(* IEC 61131-3 sources: etrolProject/分输站, 3 files *)

(* ---- com1tx.ST ---- *)
PROGRAM com1tx
VAR_EXTERNAL

END_VAR

VAR_GLOBAL

END_VAR

VAR
i		   :  UINT;
ai0_val    :  REAL :=0.0;
ai1_val    :  REAL :=0.0;
ai2_val    :  REAL :=0.0;
ai3_val    :  REAL :=0.0;
ai4_val    :  REAL :=0.0;
ai5_val    :  REAL :=0.0;
ai6_val    :  REAL :=0.0;
ai7_val    :  REAL :=0.0;
ai8_val    :  REAL :=0.0;
ai9_val    :  REAL :=0.0;
ai10_val    :  REAL :=0.0;
ai11_val    :  REAL :=0.0;
addr_val	:  UINT;
button AT %I0.0		:	BOOL;
blinker AT %Q0.6 	:	BOOL;
adr_var : UINT;
val_var : UINT;
lock_var : UINT := 0;
duishe_var : UINT := 0;
jinkoup_var : REAL;
chukoup_var : REAL;
huanrewd_var : REAL;

REG_W_UINT_VAR : REG_W_UINT;
REG_R_UINT_VAR : REG_R_UINT;
REG_MOVE_VAR   : REG_MOVE;
REG_R_REAL_VAL : REG_R_REAL;
REG_W_REAL_VAL : REG_W_REAL;
END_VAR
(*压变，温变采集*)

addr_val := 30017;
REG_R_REAL_VAL(ADDR := addr_val, SWAP := 0);
ai0_val := (REG_R_REAL_VAL.DATA - 4.0)/16.0 * 10000.0;
addr_val := 40001;
REG_W_REAL_VAL(ADDR := addr_val, SWAP := 0, DATA := ai0_val);

addr_val := 30019;
REG_R_REAL_VAL(ADDR := addr_val, SWAP := 0);
ai0_val := (REG_R_REAL_VAL.DATA - 4.0)/16.0 * 120.0 - 40.0;
addr_val := 40003;
REG_W_REAL_VAL(ADDR := addr_val, SWAP := 0, DATA := ai0_val);

addr_val := 30021;
REG_R_REAL_VAL(ADDR := addr_val, SWAP := 0);
ai0_val := (REG_R_REAL_VAL.DATA - 4.0)/16.0 * 6000.0;
addr_val := 40005;
REG_W_REAL_VAL(ADDR := addr_val, SWAP := 0, DATA := ai0_val);

addr_val := 30023;
REG_R_REAL_VAL(ADDR := addr_val, SWAP := 0);
ai0_val := (REG_R_REAL_VAL.DATA - 4.0)/16.0 * 6000.0;
addr_val := 40007;
REG_W_REAL_VAL(ADDR := addr_val, SWAP := 0, DATA := ai0_val);

addr_val := 30025;
REG_R_REAL_VAL(ADDR := addr_val, SWAP := 0);
ai0_val := (REG_R_REAL_VAL.DATA - 4.0)/16.0 * 6000.0;
addr_val := 40009;
REG_W_REAL_VAL(ADDR := addr_val, SWAP := 0, DATA := ai0_val);

addr_val := 30027;
REG_R_REAL_VAL(ADDR := addr_val, SWAP := 0);
ai0_val := (REG_R_REAL_VAL.DATA - 4.0)/16.0 * 6000.0;
addr_val := 40011;
REG_W_REAL_VAL(ADDR := addr_val, SWAP := 0, DATA := ai0_val);

addr_val := 30029;
REG_R_REAL_VAL(ADDR := addr_val, SWAP := 0);
ai0_val := (REG_R_REAL_VAL.DATA - 4.0)/16.0 * 6000.0;
addr_val := 40013;
REG_W_REAL_VAL(ADDR := addr_val, SWAP := 0, DATA := ai0_val);

addr_val := 30031;
REG_R_REAL_VAL(ADDR := addr_val, SWAP := 0);
ai0_val := (REG_R_REAL_VAL.DATA - 4.0)/16.0 * 120.0 - 40.0;
addr_val := 40015;
REG_W_REAL_VAL(ADDR := addr_val, SWAP := 0, DATA := ai0_val);

addr_val := 30033;
REG_R_REAL_VAL(ADDR := addr_val, SWAP := 0);
ai0_val := (REG_R_REAL_VAL.DATA - 4.0)/16.0 * 100.0;
addr_val := 40089;
REG_W_REAL_VAL(ADDR := addr_val, SWAP := 0, DATA := ai0_val);

addr_val := 30035;
REG_R_REAL_VAL(ADDR := addr_val, SWAP := 0);
ai0_val := (REG_R_REAL_VAL.DATA - 4.0)/16.0 * 100.0;
addr_val := 40101;
REG_W_REAL_VAL(ADDR := addr_val, SWAP := 0, DATA := ai0_val);

addr_val := 30037;
REG_R_REAL_VAL(ADDR := addr_val, SWAP := 0);
ai0_val := (REG_R_REAL_VAL.DATA - 4.0)/16.0 * 100.0;
addr_val := 40017;
REG_W_REAL_VAL(ADDR := addr_val, SWAP := 0, DATA := ai0_val);

addr_val := 30039;
REG_R_REAL_VAL(ADDR := addr_val, SWAP := 0);
ai0_val := (REG_R_REAL_VAL.DATA - 4.0)/16.0 * 100.0;
addr_val := 40019;
REG_W_REAL_VAL(ADDR := addr_val, SWAP := 0, DATA := ai0_val);

addr_val := 30041;
REG_R_REAL_VAL(ADDR := addr_val, SWAP := 0);
ai0_val := (REG_R_REAL_VAL.DATA - 4.0)/16.0 * 500.0;
addr_val := 40115;
REG_W_REAL_VAL(ADDR := addr_val, SWAP := 0, DATA := ai0_val);

END_PROGRAM

(* ---- DIANJIARE.ST ---- *)
PROGRAM DIANJIARE
VAR_EXTERNAL

END_VAR

VAR_GLOBAL

END_VAR

VAR
blinker AT %Q0.0 	:	BOOL;
blinker2 AT %Q0.1 	:	BOOL;
blinker3 AT %Q0.2   :   BOOL;
blinker4 AT %Q0.3   :   BOOL;
blinker5 AT %Q0.4   :   BOOL;
blinker6 AT %Q0.5   :   BOOL;
blinker7 AT %Q0.6   :   BOOL;
blinker8 AT %Q0.7   :   BOOL;
blinker9 AT %Q1.0   :   BOOL;
blinker10 AT %Q1.1   :   BOOL;
blinker11 AT %Q1.2   :   BOOL;
blinker12 AT %Q1.3   :   BOOL;
blinker13 AT %Q1.4   :   BOOL;
jtbutton : uint;
sgbj : uint;
i : uint;
j : uint;
kdw : uint;
gdw :uint;
kdw2 : uint;
gdw2 :uint;
kdw3 : uint;
gdw3 :uint;
kdw4 : uint;
gdw4 :uint;
jt_gdw1 : uint;
jt_gdw2 : uint;
jt_kdw1 : uint;
jt_kdw2 : uint;
addr_val : uint;
wds_val : REAL;
wdx_val : REAL;
wd_val : REAL;
par_var : uint;
lock_var : uint;
jf_open : uint;
jf_close : uint;
jf2_open : uint;
jf2_close : uint;
jf3_open : uint;
jf3_close : uint;
jf4_open : uint;
jf4_close : uint;
szd_var : uint;
REG_W_UINT_VAR : REG_W_UINT;
REG_R_UINT_VAR : REG_R_UINT;
REG_MOVE_VAR   : REG_MOVE;
REG_R_REAL_VAL : REG_R_REAL;
REG_W_REAL_VAL : REG_W_REAL;
END_VAR

REG_R_UINT_VAR(ADDR := 10018);
jtbutton := REG_R_UINT_VAR.DATA;
(*急停未按下，阀门操作*)
IF jtbutton=0 THEN
	blinker3 := TRUE;
	blinker9 := FALSE;
	blinker12 := FALSE;
	(*判断进站气液联动阀是否已修改*)
	REG_R_UINT_VAR(ADDR := 40074);
	par_var := REG_R_UINT_VAR.DATA;
	IF par_var=1 THEN
	(*参数修改*)
		REG_W_UINT_VAR(ADDR := 40074, DATA := 0);
		REG_R_UINT_VAR(ADDR := 40071);
		jf_open := REG_R_UINT_VAR.DATA;
		IF jf_open=1 THEN
			blinker := TRUE;
		ELSE
			blinker := FALSE;

		END_IF;

		REG_R_UINT_VAR(ADDR := 40072);
		jf_close := REG_R_UINT_VAR.DATA;
		IF jf_close=1 THEN
			blinker2 := TRUE;
		ELSE
			blinker2 := FALSE;
		END_IF;
	ELSE
	(*参数未修改*)
		;
	END_IF;

	REG_R_UINT_VAR(ADDR := 10003);
	kdw := REG_R_UINT_VAR.DATA;
	IF kdw=1 THEN
		blinker := FALSE;
	ELSE
		;
	END_IF;

	REG_R_UINT_VAR(ADDR := 10004);
	gdw := REG_R_UINT_VAR.DATA;
	IF gdw=1 THEN
		blinker2 := FALSE;
	ELSE
		;
	END_IF;
	(*出站电动阀*)
	REG_R_UINT_VAR(ADDR := 40078);
	par_var := REG_R_UINT_VAR.DATA;
	IF par_var=1 THEN
	(*参数修改*)
		REG_W_UINT_VAR(ADDR := 40078, DATA := 0);
		REG_R_UINT_VAR(ADDR := 40075);
		jf2_open := REG_R_UINT_VAR.DATA;
		IF jf2_open=1 THEN
			blinker4 := TRUE;
		ELSE
			blinker4 := FALSE;

		END_IF;

		REG_R_UINT_VAR(ADDR := 40076);
		jf2_close := REG_R_UINT_VAR.DATA;
		IF jf2_close=1 THEN
			blinker5 := TRUE;
		ELSE
			blinker5 := FALSE;
		END_IF;
	ELSE
	(*参数未修改*)
		;
	END_IF;

	REG_R_UINT_VAR(ADDR := 10006);
	kdw2 := REG_R_UINT_VAR.DATA;
	IF kdw2=1 THEN
		blinker4 := FALSE;
	ELSE
		;
	END_IF;

	REG_R_UINT_VAR(ADDR := 10007);
	gdw2 := REG_R_UINT_VAR.DATA;
	IF gdw2=1 THEN
		blinker5 := FALSE;
	ELSE
		;
	END_IF;

	(*进站放空阀*)
	REG_R_UINT_VAR(ADDR := 40082);
	par_var := REG_R_UINT_VAR.DATA;
	IF par_var=1 THEN
	(*参数修改*)
		REG_W_UINT_VAR(ADDR := 40082, DATA := 0);
		REG_R_UINT_VAR(ADDR := 40079);
		jf3_open := REG_R_UINT_VAR.DATA;
		IF jf3_open=1 THEN
			blinker7 := TRUE;
		ELSE
			blinker7 := FALSE;

		END_IF;

		REG_R_UINT_VAR(ADDR := 40080);
		jf3_close := REG_R_UINT_VAR.DATA;
		IF jf3_close=1 THEN
			blinker8 := TRUE;
		ELSE
			blinker8 := FALSE;
		END_IF;
	ELSE
	(*参数未修改*)
		;
	END_IF;

	REG_R_UINT_VAR(ADDR := 10010);
	kdw3 := REG_R_UINT_VAR.DATA;
	IF kdw3=1 THEN
		blinker7 := FALSE;
	ELSE
		;
	END_IF;

	REG_R_UINT_VAR(ADDR := 10011);
	gdw3 := REG_R_UINT_VAR.DATA;
	IF gdw3=1 THEN
		blinker8 := FALSE;
	ELSE
		;
	END_IF;

	(*出站放空阀*)
	REG_R_UINT_VAR(ADDR := 40086);
	par_var := REG_R_UINT_VAR.DATA;
	IF par_var=1 THEN
	(*参数修改*)
		REG_W_UINT_VAR(ADDR := 40086, DATA := 0);
		REG_R_UINT_VAR(ADDR := 40083);
		jf4_open := REG_R_UINT_VAR.DATA;
		IF jf4_open=1 THEN
			blinker10 := TRUE;
		ELSE
			blinker10 := FALSE;

		END_IF;

		REG_R_UINT_VAR(ADDR := 40084);
		jf4_close := REG_R_UINT_VAR.DATA;
		IF jf4_close=1 THEN
			blinker11 := TRUE;
		ELSE
			blinker11 := FALSE;
		END_IF;
	ELSE
	(*参数未修改*)
		;
	END_IF;

	REG_R_UINT_VAR(ADDR := 10014);
	kdw4 := REG_R_UINT_VAR.DATA;
	IF kdw4=1 THEN
		blinker10 := FALSE;
	ELSE
		;
	END_IF;

	REG_R_UINT_VAR(ADDR := 10015);
	gdw4 := REG_R_UINT_VAR.DATA;
	IF gdw4=1 THEN
		blinker11 := FALSE;
	ELSE
		;
	END_IF;
ELSE
	(*急停关阀操作*)
	(*先关进站气液，出站电动，再开进出放空*)
	blinker3 := FALSE;
	blinker9 := TRUE;
	blinker12 := TRUE;
	REG_R_UINT_VAR(ADDR := 10004);
	jt_gdw1 := REG_R_UINT_VAR.DATA;
(*	IF jt_gdw1=1 THEN
		blinker2 := FALSE;
	ELSE
		blinker2 := TRUE;
	END_IF;
	*)
	REG_R_UINT_VAR(ADDR := 10007);
	jt_gdw2 := REG_R_UINT_VAR.DATA;
	IF jt_gdw2=1 THEN
		blinker5 := FALSE;
	ELSE
		blinker5 := TRUE;
	END_IF;

	IF jt_gdw1=1 AND jt_gdw2=1 THEN
		(*REG_R_UINT_VAR(ADDR := 10010);
		jt_kdw1 := REG_R_UINT_VAR.DATA;
		IF jt_kdw1=1 THEN
			blinker7 := FALSE;
		ELSE
			blinker7 := TRUE;
		END_IF;

		REG_R_UINT_VAR(ADDR := 10014);
		jt_kdw2 := REG_R_UINT_VAR.DATA;
		IF jt_kdw2=1 THEN
			blinker10 := FALSE;
		ELSE
			blinker10 := TRUE;
		END_IF;*)
		;
	ELSE
		;
	END_IF;
END_IF;

REG_R_UINT_VAR(ADDR := 40112);
par_var := REG_R_UINT_VAR.DATA;
IF par_var=1 THEN
	REG_W_UINT_VAR(ADDR := 40112, DATA := 0);
	REG_R_UINT_VAR(ADDR := 40111);
	sgbj := REG_R_UINT_VAR.DATA;
	IF sgbj=1 THEN
		blinker13 := TRUE;
	ELSE
		blinker13 := FALSE;
	END_IF;
ELSE
	;
END_IF;
END_PROGRAM

(* ---- RX1.ST ---- *)
PROGRAM RX1
VAR_EXTERNAL
jiachou : udint;
flow_val : REAL;
start_val : uint;

END_VAR

VAR_GLOBAL
jiachou1 : udint:=0;
END_VAR

VAR
tjf_ya1_val : uint;
tjf2_ya1_val : uint;
tjf_kd1_val : uint;
tjf_ya2_val : uint;
tjf_kd2_val : uint;
i : uint;
j : uint;
blinker AT %Q0.4 	:	BOOL;
djr_start AT %Q1.5  :   BOOL;
djr_stop  AT %Q1.6  :   BOOL;
djr_par : uint;
dir_mode : uint;
dir_temp : uint;
djr_qd   : uint;
djr_tz   : uint;
djr_settemp : REAL;
dir_settemp_val : uint;
dir_fktemp : uint;
jiachounew : udint;
par_var :uint;
lock_var : uint;
szd_var	:uint;
addr_val : uint;
shunshi_val : REAL;
tongji_val : REAL;
sdyl : REAL;
sdyl_val :uint;
sdyl1 : REAL;
sdyl1_val :uint;
tjf1_qd : uint;
ai0_val : REAL;
tjf_mode :uint;
tjf2_mode :uint;
sd_fw : REAL;
sd_fw_val : uint;
sd2_fw : REAL;
sd2_fw_val : uint;
tjf_xg : uint;
tjf2_xg :uint;
REG_W_UINT_VAR : REG_W_UINT;
REG_R_UINT_VAR : REG_R_UINT;
REG_MOVE_VAR   : REG_MOVE;
REG_R_REAL_VAL : REG_R_REAL;
REG_W_REAL_VAL : REG_W_REAL;
Timer : TON;
END_VAR

(* Variable definition *)
VAR

    clear_all : PID_CLEAR_ALL;

    adr_cfg : PID_ADDR_CFG;

    adr_q : BOOL;

    val_cfg : PID_PARA_SET;

    val_q : BOOL;

    ena : PID_ENABLE;

    ena_q : BOOL;

    state : PID_AUTO;

    state_q : BOOL;

END_VAR

(*调节阀1控制*)
REG_R_UINT_VAR(ADDR := 40097);
tjf_mode := REG_R_UINT_VAR.DATA;
REG_R_UINT_VAR(ADDR := 40098);
tjf_xg := REG_R_UINT_VAR.DATA;
IF tjf_xg=1 THEN
	REG_W_UINT_VAR(ADDR := 40098, DATA := 0);
	addr_val := 40095;
	REG_R_REAL_VAL(ADDR := addr_val, SWAP := 0);
	sd_fw := (REG_R_REAL_VAL.DATA)/100.0 * 40000.0 + 10000.0;
	sd_fw_val := REAL_TO_uint(sd_fw);
	REG_W_UINT_VAR(ADDR := 40200, DATA := sd_fw_val);
END_IF;

REG_R_UINT_VAR(ADDR := 40097);
tjf_mode := REG_R_UINT_VAR.DATA;
REG_W_UINT_VAR(ADDR := 40091, DATA := tjf_mode);

addr_val := 40005;
REG_R_REAL_VAL(ADDR := addr_val, SWAP := 0);
ai0_val := REG_R_REAL_VAL.DATA;
addr_val := 40087;
REG_W_REAL_VAL(ADDR := addr_val, SWAP := 0, DATA := ai0_val);

(*调节阀2控制*)
REG_R_UINT_VAR(ADDR := 40109);
tjf2_mode := REG_R_UINT_VAR.DATA;
REG_R_UINT_VAR(ADDR := 40110);
tjf2_xg := REG_R_UINT_VAR.DATA;
IF tjf2_xg=1 THEN
	REG_W_UINT_VAR(ADDR := 40110, DATA := 0);
	addr_val := 40107;
	REG_R_REAL_VAL(ADDR := addr_val, SWAP := 0);
	sd2_fw := (REG_R_REAL_VAL.DATA)/100.0 * 40000.0 + 10000.0;
	sd2_fw_val := REAL_TO_uint(sd2_fw);
	REG_W_UINT_VAR(ADDR := 40201, DATA := sd2_fw_val);
END_IF;

REG_R_UINT_VAR(ADDR := 40109);
tjf_mode := REG_R_UINT_VAR.DATA;
REG_W_UINT_VAR(ADDR := 40103, DATA := tjf_mode);

addr_val := 40007;
REG_R_REAL_VAL(ADDR := addr_val, SWAP := 0);
ai0_val := REG_R_REAL_VAL.DATA;
addr_val := 40099;
REG_W_REAL_VAL(ADDR := addr_val, SWAP := 0, DATA := ai0_val);

(*电加热*)
REG_R_UINT_VAR(ADDR := 40121);
djr_par := REG_R_UINT_VAR.DATA;
IF djr_par=1 THEN
	REG_W_UINT_VAR(ADDR := 40121, DATA := 0);
	REG_R_UINT_VAR(ADDR := 40117);
	djr_qd := REG_R_UINT_VAR.DATA;
	IF djr_qd=1 THEN
		djr_start := TRUE;
		REG_R_REAL_VAL(ADDR := 40119, SWAP := 0);
		djr_settemp := (REG_R_REAL_VAL.DATA)/500.0 * 40000.0 + 10000.0;
		dir_settemp_val := REAL_TO_uint(djr_settemp);
		REG_W_UINT_VAR(ADDR := 40304, DATA := dir_settemp_val);
		(*REG_R_UINT_VAR(ADDR := 30013);
		dir_fktemp := REG_R_UINT_VAR.DATA;
		REG_W_UINT_VAR(ADDR := 40305, DATA := dir_fktemp);*)
	ELSE
		djr_start := FALSE;
	END_IF;

	REG_R_UINT_VAR(ADDR := 40118);
	djr_tz := REG_R_UINT_VAR.DATA;
	IF djr_tz=1 THEN
		djr_stop := TRUE;
	ELSE
		djr_stop := FALSE;
	END_IF;

END_IF;

END_PROGRAM
